FUNCTION NextMinorStep : UDINT
VAR_INPUT
	StateVar	: UDINT;
END_VAR
VAR
END_VAR

NextMinorStep := StateVar + 1;

END_FUNCTION

(* stored: Version 1.1.0.1, ProductVersion 3.1.4024.12
   POU NextMinorStep: Id {70ffbba5-aa46-4222-be25-7aac3270a8dc}, SpecialFunc None *)
